// TIA Portal V18 export
DATA_BLOCK "Utility_PID_DB_1"   // DB197
VERSION : 0.1
// stored: AutoNumber true, DBAccessibleFromOPCUA true, DBAccessibleFromWebserver true, InstanceOfName Utility_PID, InstanceOfType FB
"Utility_PID"
   // VAR_INPUT
   //    START : Bool;
   //    SP : Real;
   //    PV : Real;
   //    CONTROL_MODE : Int;
   //    "TIME" : Int;
   //    PRE_SP : Int;
   //    AM : Bool;
   //    P : Int;
   //    I : Int;
   //    D : Int;
   //    JAC_IN : Real;
   //    JAC_OUT : Real;
   //    HHSP : Real;
   //    HSP : Real;
   //    LSP : Real;
   //    LLSP : Real;
   //    PIDRST : Bool;
   //    SOURCE_SEL : Int;
   //    AIR_XV_OPN : Bool;
   //    BYP_XV_OPN : Bool;
   //    VENT_OPN : Bool;
   //    CONDENSATE_XV_OPN : Bool;
   //    DRAIN_XV_OPN : Bool;
   //    SCV_XV_OPN : Bool;
   // END_VAR
   // VAR_OUTPUT
   //    START_PV : Real;
   //    CVOUT : Int;
   //    SCVOUT : Real;
   //    STATUS : Int;
   //    RAMP_SP : Real;
   //    JSP : Real;
   //    PID_PV : Real;
   //    RUN_MIN : Int;
   //    RUN_HR : Int;
   //    STEAM_SCVOUT : Real;
   //    STEAM_CVOUT : Int;
   // END_VAR
   // VAR_IN_OUT
   //    PAUSE : Bool;
   //    MAN_OUT : Real;
   //    TEMP_LIMIT : Real;
   //    STEAM_MAN_OUT : Real;
   // END_VAR
   // VAR
   //    RAMP_MODE : Bool;
   //    MAINT_MODE : Bool;
   //    J_MAINT_MODE : Bool;
   //    NO_RAMP : Bool;
   //    HEAT_COOL : Bool;
   //    BSTBIT : Bool;
   //    HOLD : Int;
   //    RAMP : Real;
   //    RAMP_RST : Bool;
   //    RMPSTART : Bool;
   //    Ramp_Substitute : Real;
   //    RAMP_INIT_RST : Bool;
   //    JKT_RAMP : Bool;
   //    MASS_CONTROL : Bool;
   //    TIMER_TRIG : Bool;
   //    iSTEAM_SCVOUT : Real;
   //    iSTEAM_CVOUT : Int;
   //    iSTEAM_SCV_SCL : Real;
   //    iSTEAM_CV_SCL : Int;
   //    iDRAIN_UP : Bool;
   // END_VAR
BEGIN
END_DATA_BLOCK
